FUNCTION_BLOCK FuncGeneralesMultidisc1
VAR_INPUT

	
END_VAR
VAR_OUTPUT	
	s_ModeloActualTabla:STRING;
	s_ModeloEleccionTabla:STRING;
	s_JustificaParoComun:STRING;
	s_FechaInicModeloTab:STRING;
END_VAR
VAR
	Reset_Fin_Prod:BOOL;
	P_FinProduccion:BOOL;
	P_EscribirModelo:BOOL;
	sModeloEleccionTabla:STRING;
	pul_Justif_Paro:BOOL;
END_VAR
VAR PERSISTENT 

END_VAR

//                             >>>>>>>>>>>>>>>> Modelo de la tabla <<<<<<<<<<<<<<<<<

//Fin de producción 		
IF P_FinProduccion THEN 
Fin_Produccion();
END_IF;
IF P_EscribirModelo THEN 
	Inicio_Nuevo_Modelo();
END_IF


Direccionamiento_variables_com();

ACTION Direccionamiento_variables_com:
	//                           	>>>>>>>>>>>>>>>>>>>>>>>>>>>>      STRING  <<<<<<<<<<<<<<<<<<<<<<<<<<<<<<<<
    Var_Com_CH4_MulDis.aStringCom[80] := s_ModeloActualTabla;
	Var_Com_CH4_MulDis.aStringCom[81] := s_JustificaParoComun;
	Var_Com_CH4_MulDis.aStringCom[82] := s_FechaInicModeloTab;
END_ACTION

METHOD Fin_Produccion : BOOL
VAR_INPUT	
END_VAR
var
	Puls_Fin_Produccion:BOOL;	
END_VAR
//Llamada a la función de fin de producción de Corte húmedo 4
FuncParoNodoCorteH4Remote1.Funci_CortHum4.Fin_Produccion();



s_ModeloActualTabla:= 'Sin modelo de pieza';
//	FechaInicModeloTab:= 'Sin modelo de pieza';
s_ModeloEleccionTabla:= 'Sin modelo de pieza';
END_METHOD

METHOD Inicio_Nuevo_Modelo : BOOL
VAR_INPUT
END_VAR
VAR
END_VAR

// Envías la fecha de inicio modelo de tabla 
s_FechaInicModeloTab:=Fecha_PLC.Mes_Dia_Hora_Min_Real;

//Envías el modelo de la tabla de la variable preelección  
s_ModeloActualTabla:=sModeloEleccionTabla;
END_METHOD

END_FUNCTION_BLOCK

(* stored: Version 1.1.0.1, ProductVersion 3.1.4024.12
   POU FuncGeneralesMultidisc1: Id {202f2458-e1f8-4dbc-bbad-08ad70ca02eb}, SpecialFunc None
   Action Direccionamiento_variables_com: Id {832475eb-2cbd-47c0-b591-9cc7574195f8}
   Method Fin_Produccion: Id {f98c57f5-c388-4d9e-982c-a29b2c0a8627}
   Method Inicio_Nuevo_Modelo: Id {9af42117-f1fa-463c-9afb-b86795815813} *)
